Universal Robots URScript: 00C_02_JuXian.script

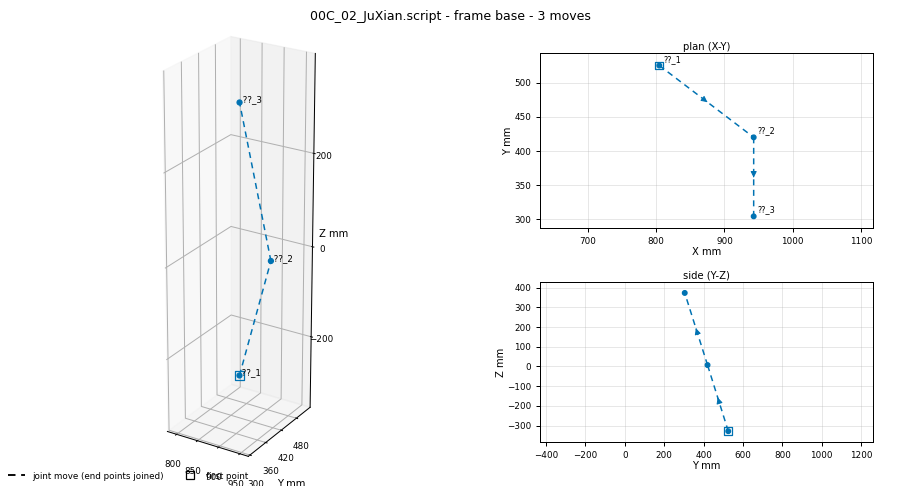
[picture p0: tool path of 00C_02_JuXian.script in frame base, 3 of 3 moves have a stored position in this frame; points joined in program order, loops and branches not executed]
def P00C_02_JuXian():
  set_standard_analog_input_domain(0, 1)
  set_standard_analog_input_domain(1, 1)
  set_tool_analog_input_domain(0, 1)
  set_tool_analog_input_domain(1, 1)
  set_analog_outputdomain(0, 0)
  set_analog_outputdomain(1, 0)
  set_tool_voltage(0)
  set_input_actions_to_default()
  set_tcp(p[-0.06448999999999999,0.0207,0.28314999999999996,0.0,0.0,1.5902])
  set_payload(8.0)
  set_safety_mode_transition_hardness(1)
  set_gravity([0.0, 0.0, 9.82])
  $ 1 "机器人程序"
  $ 2 "MoveJ"
  $ 3 "路点_1"
  set_tcp(p[-8.5E-4,0.01448,0.31003,0.0,0.0,-0.3645])
  movej(get_inverse_kin(p[.804567293087, .525319472513, -.328924413572, .111197400113, 1.481243442736, -.236017489866], qnear=[1.1887894868850708, -2.8590243498431605, -1.742481533681051, -1.1460588614093226, -0.19416314760317022, -1.8057902495013636]), a=0.6981317007977318, v=0.5235987755982988)
  $ 4 "路点_2"
  set_tcp(p[-8.5E-4,0.01448,0.31003,0.0,0.0,-0.3645])
  movej(get_inverse_kin(p[.942814963611, .420113235798, .006830243995, -.471207470381, 1.353267818753, -.663529095720], qnear=[0.8986625671386719, -2.3152812162982386, -1.985840145741598, -1.6769560019122522, -0.6309183279620569, -2.1957572142230433]), a=0.6981317007977318, v=0.5235987755982988)
  $ 5 "路点_3"
  set_tcp(p[-8.5E-4,0.01448,0.31003,0.0,0.0,-0.3645])
  movej(get_inverse_kin(p[.942797157451, .304374145277, .372975668928, -1.314426838057, .989200724266, -1.148646982301], qnear=[0.6537488698959351, -1.6546004454242151, -1.9450820128070276, -2.62942344347109, -1.1071928183185022, -2.8940122763263147]), a=0.6981317007977318, v=0.5235987755982988)
end
